{attribute 'GeneratedUsingTerminal: EL2521-0000-1019'}
{attribute addProperty BoxType "EL2521-0000-1019"}
{attribute addProperty Id "StatusAT %I*Status_CDD96F355Counter_valueAT %I*UINT2"}
{attribute addProperty CRC "56910025"}
{attribute addProperty Size "7"}
TYPE ENC_Status_compact_036460C9 :
STRUCT
	{attribute addProperty Name "Status"}
	Status AT %I* : Status_CDD96F35;
	{attribute addProperty Name "Counter_value"}
	Counter_value AT %I* : UINT;
END_STRUCT
END_TYPE

(* stored: Version 1.2.0.0, ProductVersion 3.1.4024.9
   DUT ENC_Status_compact_036460C9: Id {e65bd35b-5589-4086-9ed8-101e1c97cd0a} *)
